(* IEC 61131-3 sources: com.logicals.lc3.webinar/usRTS_RPMControl_iSOC/src_FB_LIB_SAFE/Numeric/REAL, 8 files *)

(* ---- wADD_REAL_2.iecst ---- *)
NAMESPACE logicals.web.standard
NAMESPACE numeric

/*
 * Function block wrapper for IEC 61131-3 ADD<br>
 * IN1 =  1st value (REAL)<br>
 * IN2 =  2nd value (REAL)<br>
 * OUT = Sum of all input values (REAL)<br>
 */
FUNCTION_BLOCK wADD_REAL_2
	{ vNameAlignment:="center"; altName:="+"; bgColor:="Orange"; width:=40; hideIONames; }
	VAR_INPUT
		IN1 : REAL;
		IN2 : REAL;
	END_VAR
	VAR_OUTPUT
		OUT : REAL;
	END_VAR

	OUT := ADD(IN1:=IN1, IN2:=IN2, ENO=>ENO);
END_FUNCTION_BLOCK

END_NAMESPACE
END_NAMESPACE

(* ---- wADD_REAL_3.iecst ---- *)
NAMESPACE logicals.web.standard
NAMESPACE numeric

/*
 * Function block wrapper for IEC 61131-3 ADD<br>
 * IN1 =  1st value (REAL)<br>
 * IN2 =  2nd value (REAL)<br>
 * IN3 =  3rd value (REAL)<br>
 * OUT = Sum of all input values (REAL)<br>
 */
FUNCTION_BLOCK wADD_REAL_3
	{ vNameAlignment:="center"; altName:="+"; bgColor:="Orange"; width:=40; hideIONames; }
	VAR_INPUT
		IN1 : REAL;
		IN2 : REAL;
		IN3 : REAL;
	END_VAR
	VAR_OUTPUT
		OUT : REAL;
	END_VAR

	OUT := ADD(IN1:=IN1, IN2:=IN2, IN3:=IN3, ENO=>ENO);
END_FUNCTION_BLOCK

END_NAMESPACE
END_NAMESPACE

(* ---- wADD_REAL_4.iecst ---- *)
NAMESPACE logicals.web.standard
NAMESPACE numeric

/*
 * Function block wrapper for IEC 61131-3 ADD<br>
 * IN1 =  1st value (REAL)<br>
 * IN2 =  2nd value (REAL)<br>
 * IN3 =  3rd value (REAL)<br>
 * IN4 =  4th value (REAL)<br>
 * OUT = Sum of all input values (REAL)<br>
 */
FUNCTION_BLOCK wADD_REAL_4
	{ vNameAlignment:="center"; altName:="+"; bgColor:="Orange"; width:=40; hideIONames; }
	VAR_INPUT
		IN1 : REAL;
		IN2 : REAL;
		IN3 : REAL;
		IN4 : REAL;
	END_VAR
	VAR_OUTPUT
		OUT : REAL;
	END_VAR

	OUT := ADD(IN1:=IN1, IN2:=IN2, IN3:=IN3, IN4:=IN4, ENO=>ENO);
END_FUNCTION_BLOCK

END_NAMESPACE
END_NAMESPACE

(* ---- wDIV_REAL.iecst ---- *)
NAMESPACE logicals.web.standard
NAMESPACE numeric

/*
 * Function block wrapper for IEC 61131-3 DIV<br>
 * IN1 =  1st value (REAL)<br>
 * IN2 =  2nd value (REAL)<br>
 * OUT = quotient of IN1 divided by IN2 (REAL)<br>
 */
FUNCTION_BLOCK wDIV_REAL
	{ vNameAlignment:="center"; altName:="/"; bgColor:="Orange"; width:=40; hideIONames; }
	VAR_INPUT
		IN1 : REAL;
		IN2 : REAL;
	END_VAR
	VAR_OUTPUT
		OUT : REAL;
	END_VAR

	OUT := DIV(IN1:=IN1, IN2:=IN2, ENO=>ENO);
END_FUNCTION_BLOCK

END_NAMESPACE
END_NAMESPACE

(* ---- wMUL_REAL_2.iecst ---- *)
NAMESPACE logicals.web.standard
NAMESPACE numeric

/*
 * Function block wrapper for IEC 61131-3 MUL<br>
 * IN1 =  1st value (REAL)<br>
 * IN2 =  2nd value (REAL)<br>
 * OUT = Product of multiplication of all inputs (REAL)<br>
 */
FUNCTION_BLOCK wMUL_REAL_2
	{ vNameAlignment:="center"; altName:="*"; bgColor:="Orange"; width:=40; hideIONames; }
	VAR_INPUT
		IN1 : REAL;
		IN2 : REAL;
	END_VAR
	VAR_OUTPUT
		OUT : REAL;
	END_VAR

	OUT := MUL(IN1:=IN1, IN2:=IN2, ENO=>ENO);
END_FUNCTION_BLOCK

END_NAMESPACE
END_NAMESPACE

(* ---- wMUL_REAL_3.iecst ---- *)
NAMESPACE logicals.web.standard
NAMESPACE numeric

/*
 * Function block wrapper for IEC 61131-3 MUL<br>
 * IN1 =  1st value (REAL)<br>
 * IN2 =  2nd value (REAL)<br>
 * IN3 =  3rd value (REAL)<br>
 * OUT = Product of multiplication of all inputs (REAL)<br>
 */
FUNCTION_BLOCK wMUL_REAL_3
	{ vNameAlignment:="center"; altName:="*"; bgColor:="Orange"; width:=40; hideIONames; }
	VAR_INPUT
		IN1 : REAL;
		IN2 : REAL;
		IN3 : REAL;
	END_VAR
	VAR_OUTPUT
		OUT : REAL;
	END_VAR

	OUT := MUL(IN1:=IN1, IN2:=IN2, IN3:=IN3, ENO=>ENO);
END_FUNCTION_BLOCK

END_NAMESPACE
END_NAMESPACE

(* ---- wMUL_REAL_4.iecst ---- *)
NAMESPACE logicals.web.standard
NAMESPACE numeric

/*
 * Function block wrapper for IEC 61131-3 MUL<br>
 * IN1 =  1st value (REAL)<br>
 * IN2 =  2nd value (REAL)<br>
 * IN3 =  3rd value (REAL)<br>
 * IN4 =  4th value (REAL)<br>
 * OUT = Product of multiplication of all inputs (REAL)<br>
 */
FUNCTION_BLOCK wMUL_REAL_4
	{ vNameAlignment:="center"; altName:="*"; bgColor:="Orange"; width:=40; hideIONames; }
	VAR_INPUT
		IN1 : REAL;
		IN2 : REAL;
		IN3 : REAL;
		IN4 : REAL;
	END_VAR
	VAR_OUTPUT
		OUT : REAL;
	END_VAR

	OUT := MUL(IN1:=IN1, IN2:=IN2, IN3:=IN3, IN4:=IN4, ENO=>ENO);
END_FUNCTION_BLOCK

END_NAMESPACE
END_NAMESPACE

(* ---- wSUB_REAL.iecst ---- *)
NAMESPACE logicals.web.standard
NAMESPACE numeric

/*
 * Function block wrapper for IEC 61131-3 SUB<br>
 * IN1 =  1st value (REAL)<br>
 * IN2 =  2nd value (REAL)<br>
 * OUT = IN1 minus IN2 (REAL)<br>
 */
FUNCTION_BLOCK wSUB_REAL
	{ vNameAlignment:="center"; altName:="-"; bgColor:="Orange"; width:=40; hideIONames; }
	VAR_INPUT
		IN1 : REAL;
		IN2 : REAL;
	END_VAR
	VAR_OUTPUT
		OUT : REAL;
	END_VAR

	OUT := SUB(IN1:=IN1, IN2:=IN2, ENO=>ENO);
END_FUNCTION_BLOCK

END_NAMESPACE
END_NAMESPACE
